INTERFACE ITF_BaseMessengerSender

END_INTERFACE

(* stored: Version 1.1.0.1
   Itf ITF_BaseMessengerSender: Id {f2c748b8-07c6-03cf-04c2-0bcc78ff32eb} *)
